{attribute 'Tc2GvlVarNames'}
VAR_CONFIG
END_VAR

(* stored: Version 1.1.0.1, ProductVersion 3.1.4024.15
   GVL Variable_Configuration: Id {29a7d9e6-d143-4841-96c2-77bac407c8ae} *)
